FUNCTION_BLOCK FB_Uint_Udint
VAR
	nOldValue: UINT;
	nDiff: DINT;
	nMinus: BOOL;
	nPlus: BOOL;
END_VAR
VAR_INPUT
	nInSmall: UINT;
END_VAR

VAR_IN_OUT
	nBig: UDINT;
END_VAR

nDiff := nInSmall - nOldValue;


(* Richtung Minus *)
IF ndiff > 10000 THEN
	nBig := nBig - 1;
	nMinus := TRUE;
END_IF

(* Richtung Plus *)
IF ndiff < -10000 THEN
	nBig := nBig + 1;
	nPlus := TRUE;
END_IF

IF (ndiff < 500) AND ndiff > -500 THEN
  nBig := DINT_TO_UDINT( UDINT_TO_DINT(nBig) + nDiff) ;
END_IF
nOldValue := nInSmall;

END_FUNCTION_BLOCK

(* stored: Version 1.1.0.1, ProductVersion 3.1.4019.2
   POU FB_Uint_Udint: Id {ea86ec42-82de-47d3-a502-3c3c1a29a03f}, SpecialFunc None *)
